TYPE ST_SYSTEM_SoftwareVersion :
STRUCT
	sPLCVersionHMI					: STRING;
	sScreenVersionInfoHMI				: STRING;
	sBridgeVersionHMI					: STRING;
END_STRUCT
END_TYPE

(* stored: Version 1.1.0.1
   DUT ST_SYSTEM_SoftwareVersion: Id {7591316a-6db5-4e7b-a133-ab34a4ff1cdb} *)
